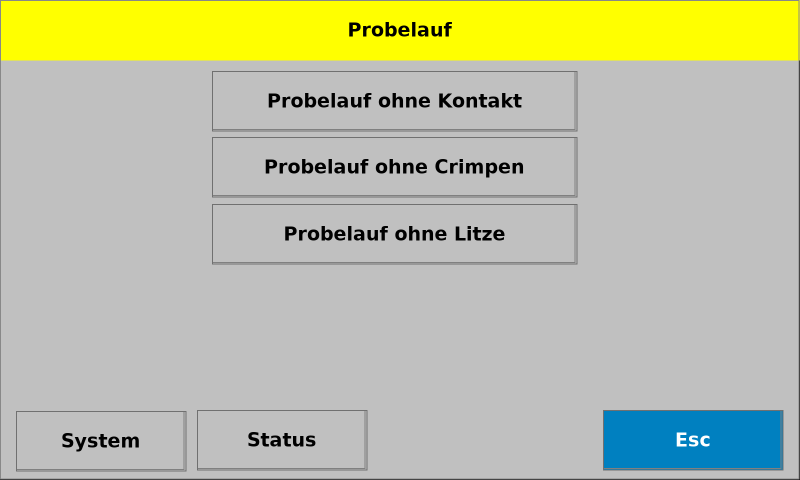
VISUALIZATION Probelauf  // 800x480
    Rectangle (0,0 800x480)
    Rectangle (0,0 800x60), "Probelauf"
    Button (212,71 365x60), "Probelauf ohne Kontakt", colour toggle: VAT.bProbelOhneKontakt
        toggle VAT.bProbelOhneKontakt
        OnMouseClick: execute { F_AuswertungBefehlstastenVonTP(tastenWert := CVL.PROBE_OHNE_KONT); }
    Button (212,137 365x60), "Probelauf ohne Crimpen", colour toggle: VAT.bProbelOhneCrimpen
        toggle VAT.bProbelOhneCrimpen
        OnMouseClick: execute { F_AuswertungBefehlstastenVonTP(tastenWert := CVL.PROBE_OHNE_CRIMP); }
    Button (212,204 365x60), "Probelauf ohne Litze", colour toggle: VAT.bProbelOhneLitze
        toggle VAT.bProbelOhneCrimpen
        OnMouseClick: execute { F_AuswertungBefehlstastenVonTP(tastenWert := CVL.PROBE_OHNE_LITZE); }
    Button (16,411 170x60), "System"
        tap P_HmiHandling.bClose
    Button (197,410 170x60), "Status"
    Button (603,410 180x60), "Esc"
        OnMouseUp: change screen: Previous 
END_VISUALIZATION

(* stored: Version 1.1.0.1, ProductVersion 3.1.4024.3
   Visu Probelauf: Id {24b10917-44f0-4ab4-8346-879dfe80cfb9} *)
